Staubli VAL3: toJointDeg.pgx

public program toJointDeg(num& x_nJointArray[], joint& x_jJoint)
  local num l_nRad2Deg
  local num l_nM2Mm
begin
  // Copyright (c) 2016, Ocado Technology - Robotics Research Team
  //
  // Licensed under the Apache License, Version 2.0 (the "License");
  // you may not use this file except in compliance with the License.
  // You may obtain a copy of the License at
  //
  //     http://www.apache.org/licenses/LICENSE-2.0
  //
  // Unless required by applicable law or agreed to in writing, software
  // distributed under the License is distributed on an "AS IS" BASIS,
  // WITHOUT WARRANTIES OR CONDITIONS OF ANY KIND, either express or implied.
  // See the License for the specific language governing permissions and
  // limitations under the License.



  l_nRad2Deg = 57.2957795131
  l_nM2Mm = 1000

  // RS60/RS-TS-safe mapping: first three axes are revolute (rad->deg),
  // fourth axis is linear (m->mm).
  x_jJoint.j1 = x_nJointArray[0] * l_nRad2Deg
  x_jJoint.j2 = x_nJointArray[1] * l_nRad2Deg
  x_jJoint.j3 = x_nJointArray[2] * l_nRad2Deg
  x_jJoint.j4 = x_nJointArray[3] * l_nM2Mm
end
